FUNCTION_BLOCK ReadyToHaltedUnifiedProgramTransition EXTENDS ReadyToHaltedProgramTransition
VAR_STAT
	//! <summary>Class name shared by all instances of this function block.</summary>
	{attribute 'OPC.UA.DA' := '0'}
	_ClassName : STRING := __POUNAME();
END_VAR

{attribute 'monitoring' := 'call'}
PROPERTY ClassName : REFERENCE TO STRING
GET
ClassName REF= _ClassName;
END_GET
END_PROPERTY

END_FUNCTION_BLOCK

(* stored: Version 1.1.0.1
   POU ReadyToHaltedUnifiedProgramTransition: Id {5f5a6c31-5f27-4b7d-a8d0-3d26d69d9fd4}, SpecialFunc None
   Property ClassName: Id {6b007aba-a50c-4d3a-a694-368fa302c299}
   Get Get: Id {820dfd52-ccfb-4cad-a0a3-21d6bf895a1b} *)
